PROGRAM Axis04_Interlock
VAR
	Always_ON	:	BOOL	:=TRUE	;//상시 ON 
	Always_OFF	:	BOOL	:=FALSE	;//상시 OFF
END_VAR

// NETWORK 1

END_PROGRAM

(* stored: Version 1.1.0.1, ProductVersion 3.1.4024.15
   POU Axis04_Interlock: Id {e5891fc9-b3e3-4690-9819-5aa86482a7cb}, SpecialFunc None *)
